// TIA Portal V15.1 export
// export: Created 2024-05-17T05:38:13.9660072Z, ExportSetting WithDefaults, DisplayName Totally Integrated Automation Portal, DisplayVersion V15.1 Update 5, DisplayName TIA Portal Openness, DisplayVersion V15.1 Update 5, DisplayName SINAMICS Startdrive Advanced, DisplayVersion V15.1, DisplayName G130, G150, S120, S150, SINAMICS MV, S210, DisplayVersion V15.1, DisplayName G110M, G120, G120C, G120D, G120P, DisplayVersion V15.1, DisplayName STEP 7 Professional, DisplayVersion V15.1 Update 5, DisplayName STEP 7 Safety, DisplayVersion V15.1, DisplayName WinCC Professional, DisplayVersion V15.1 Update 5, DisplayName SIMATIC Visualization Architect, DisplayVersion V15.1
DATA_BLOCK "_209210ZS01PNIODiag"   // DB324
{ S7_Optimized_Access := 'FALSE' }
AUTHOR : VCC
VERSION : 0.1
// stored: AutoNumber false, DBAccessibleFromOPCUA true, IsOnlyStoredInLoadMemory false, IsWriteProtectedInAS false
   VAR RETAIN
      "AA_209210AS10-JW40" { ExternalAccessible := 'False'; ExternalVisible := 'False'; ExternalWritable := 'False'} : Bool;   // Profinet device don't exist - ET200sp I/O - Busnode 210AS10 - node 40
      "AA_209210AX01-JW41" { ExternalAccessible := 'False'; ExternalVisible := 'False'; ExternalWritable := 'False'} : Bool;   // Profinet device don't exist - ET200sp I/O - Busnode 210AX01 - node 41
      "AA_209210AS11-JW42" { ExternalAccessible := 'False'; ExternalVisible := 'False'; ExternalWritable := 'False'} : Bool;   // Profinet device don't exist - ET200sp I/O - Busnode 210AS11 - node 42
      "AA_209210AX02-JW43" { ExternalAccessible := 'False'; ExternalVisible := 'False'; ExternalWritable := 'False'} : Bool;   // Profinet device don't exist - ET200sp I/O - Busnode 210AX02 - node 43
      "AC_209210CWP10-JX44" { ExternalAccessible := 'False'; ExternalVisible := 'False'; ExternalWritable := 'False'} : Bool;   // Profinet device don't exist - ET200eco I/O - Module 210CWP10 - node 44
      "AC_209210CWP10-JX45" { ExternalAccessible := 'False'; ExternalVisible := 'False'; ExternalWritable := 'False'} : Bool;   // Profinet device don't exist - ET200eco I/O - Module 210CWP10 - node 45
      "AC_209210CWP20-JX46" { ExternalAccessible := 'False'; ExternalVisible := 'False'; ExternalWritable := 'False'} : Bool;   // Profinet device don't exist - ET200eco I/O - Module 210CWP20 - node 46
      "AC_209210CWP20-JX47" { ExternalAccessible := 'False'; ExternalVisible := 'False'; ExternalWritable := 'False'} : Bool;   // Profinet device don't exist - ET200eco I/O - Module 210CWP20 - node 47
      "AA_209210AS20-JW48" { ExternalAccessible := 'False'; ExternalVisible := 'False'; ExternalWritable := 'False'} : Bool;   // Profinet device don't exist - ET200sp I/O - Busnode 210AS20 - node 48
      "AB_209000AK03M1-UE130" { ExternalAccessible := 'False'; ExternalVisible := 'False'; ExternalWritable := 'False'} : Bool;   // Profinet device don't exist - MoviDrive - 210CR21M1 - node 130
      "AB_209000AK03M4-UE131" { ExternalAccessible := 'False'; ExternalVisible := 'False'; ExternalWritable := 'False'} : Bool;   // Profinet device don't exist - MoviDrive - 210CS22M4(Power) - node 131
      "AB_209000AK03M4-UE132" { ExternalAccessible := 'False'; ExternalVisible := 'False'; ExternalWritable := 'False'} : Bool;   // Profinet device don't exist - MoviDrive - 210CS22M4(Brake) - node 132
      "AB_209000AK03M1-UE133" { ExternalAccessible := 'False'; ExternalVisible := 'False'; ExternalWritable := 'False'} : Bool;   // Profinet device don't exist - MoviDrive - 210CR23M1 - node 133
      "AB_209210CHB21M14-UE134" { ExternalAccessible := 'False'; ExternalVisible := 'False'; ExternalWritable := 'False'} : Bool;   // Profinet device don't exist - MoviFit - 210CHB21M14 - node 134
      "AA_209210Field-JW221" { ExternalAccessible := 'False'; ExternalVisible := 'False'; ExternalWritable := 'False'} : Bool;   // Profinet device don't exist - Field Switch - Safety Zone 210 - node 221
      "AA_209210Field-JW231" { ExternalAccessible := 'False'; ExternalVisible := 'False'; ExternalWritable := 'False'} : Bool;   // Profinet device don't exist - Field Switch - Safety Zone 210 - node 231
      "AC_209210AS10-JW40Fault" { ExternalAccessible := 'False'; ExternalVisible := 'False'; ExternalWritable := 'False'} : Bool;   // Faulty profinet device -> For more detail information look for N.A. alarms in the alarmlist - ET200sp I/O - Busnode 210AS10 - node 40
      "AC_209210AX01-JW41Fault" { ExternalAccessible := 'False'; ExternalVisible := 'False'; ExternalWritable := 'False'} : Bool;   // Faulty profinet device -> For more detail information look for N.A. alarms in the alarmlist - ET200sp I/O - Busnode 210AX01 - node 41
      "AC_209210AS11-JW42Fault" { ExternalAccessible := 'False'; ExternalVisible := 'False'; ExternalWritable := 'False'} : Bool;   // Faulty profinet device -> For more detail information look for N.A. alarms in the alarmlist - ET200sp I/O - Busnode 210AS11 - node 42
      "AC_209210AX02-JW43Fault" { ExternalAccessible := 'False'; ExternalVisible := 'False'; ExternalWritable := 'False'} : Bool;   // Faulty profinet device -> For more detail information look for N.A. alarms in the alarmlist - ET200sp I/O - Busnode 210AX02 - node 43
      "AC_209210CWP10-JX44Fault" { ExternalAccessible := 'False'; ExternalVisible := 'False'; ExternalWritable := 'False'} : Bool;   // Faulty profinet device -> For more detail information look for N.A. alarms in the alarmlist - ET200eco I/O - Module 210CWP10 - node 44
      "AC_209210CWP10-JX45Fault" { ExternalAccessible := 'False'; ExternalVisible := 'False'; ExternalWritable := 'False'} : Bool;   // Faulty profinet device -> For more detail information look for N.A. alarms in the alarmlist - ET200eco I/O - Module 210CWP10 - node 45
      "AC_209210CWP20-JX46Fault" { ExternalAccessible := 'False'; ExternalVisible := 'False'; ExternalWritable := 'False'} : Bool;   // Faulty profinet device -> For more detail information look for N.A. alarms in the alarmlist - ET200eco I/O - Module 210CWP20 - node 46
      "AC_209210CWP20-JX47Fault" { ExternalAccessible := 'False'; ExternalVisible := 'False'; ExternalWritable := 'False'} : Bool;   // Faulty profinet device -> For more detail information look for N.A. alarms in the alarmlist - ET200eco I/O - Module 210CWP20 - node 47
      "AC_209210AS20-JW48Fault" { ExternalAccessible := 'False'; ExternalVisible := 'False'; ExternalWritable := 'False'} : Bool;   // Faulty profinet device -> For more detail information look for N.A. alarms in the alarmlist - ET200sp I/O - Busnode 210AS20 - node 48
      "AC_209000AK03M1-UE130Fault" { ExternalAccessible := 'False'; ExternalVisible := 'False'; ExternalWritable := 'False'} : Bool;   // Faulty profinet device -> For more detail information look for N.A. alarms in the alarmlist - MoviDrive - 210CR21M1 - node 130
      "AC_209000AK03M4-UE131Fault" { ExternalAccessible := 'False'; ExternalVisible := 'False'; ExternalWritable := 'False'} : Bool;   // Faulty profinet device -> For more detail information look for N.A. alarms in the alarmlist - MoviDrive - 210CS22M4(Power) - node 131
      "AC_209000AK03M4-UE132Fault" { ExternalAccessible := 'False'; ExternalVisible := 'False'; ExternalWritable := 'False'} : Bool;   // Faulty profinet device -> For more detail information look for N.A. alarms in the alarmlist - MoviDrive - 210CS22M4(Brake) - node 132
      "AC_209000AK03M1-UE133Fault" { ExternalAccessible := 'False'; ExternalVisible := 'False'; ExternalWritable := 'False'} : Bool;   // Faulty profinet device -> For more detail information look for N.A. alarms in the alarmlist - MoviDrive - 210CR23M1 - node 133
      "AC_209210CHB21M14-UE134Fault" { ExternalAccessible := 'False'; ExternalVisible := 'False'; ExternalWritable := 'False'} : Bool;   // Faulty profinet device -> For more detail information look for N.A. alarms in the alarmlist - MoviFit - 210CHB21M14 - node 134
      "AC_209210Field-JW221Fault" { ExternalAccessible := 'False'; ExternalVisible := 'False'; ExternalWritable := 'False'} : Bool;   // Faulty profinet device -> For more detail information look for N.A. alarms in the alarmlist - Field Switch - Safety Zone 210 - node 221
      "AC_209210Field-JW231Fault" { ExternalAccessible := 'False'; ExternalVisible := 'False'; ExternalWritable := 'False'} : Bool;   // Faulty profinet device -> For more detail information look for N.A. alarms in the alarmlist - Field Switch - Safety Zone 210 - node 231
      "209210AS10-JW40AlarmABCondition" { ExternalAccessible := 'False'; ExternalVisible := 'False'; ExternalWritable := 'False'} : Bool;   // Alarm AB condition
      "209210AX01-JW41AlarmABCondition" { ExternalAccessible := 'False'; ExternalVisible := 'False'; ExternalWritable := 'False'} : Bool;   // Alarm AB condition
      "209210AS11-JW42AlarmABCondition" { ExternalAccessible := 'False'; ExternalVisible := 'False'; ExternalWritable := 'False'} : Bool;   // Alarm AB condition
      "209210AX02-JW43AlarmABCondition" { ExternalAccessible := 'False'; ExternalVisible := 'False'; ExternalWritable := 'False'} : Bool;   // Alarm AB condition
      "209210AS20-JW48AlarmABCondition" { ExternalAccessible := 'False'; ExternalVisible := 'False'; ExternalWritable := 'False'} : Bool;   // Alarm AB condition
      "209000AK03M1-UE130AlarmABCondition" { ExternalAccessible := 'False'; ExternalVisible := 'False'; ExternalWritable := 'False'} : Bool;   // Alarm AB condition
      "209000AK03M4-UE131AlarmABCondition" { ExternalAccessible := 'False'; ExternalVisible := 'False'; ExternalWritable := 'False'} : Bool;   // Alarm AB condition
      "209000AK03M4-UE132AlarmABCondition" { ExternalAccessible := 'False'; ExternalVisible := 'False'; ExternalWritable := 'False'} : Bool;   // Alarm AB condition
      "209000AK03M1-UE133AlarmABCondition" { ExternalAccessible := 'False'; ExternalVisible := 'False'; ExternalWritable := 'False'} : Bool;   // Alarm AB condition
      "209210CHB21M14-UE134AlarmABCondition" { ExternalAccessible := 'False'; ExternalVisible := 'False'; ExternalWritable := 'False'} : Bool;   // Alarm AB condition
      "209210Field-JW221AlarmABCondition" { ExternalAccessible := 'False'; ExternalVisible := 'False'; ExternalWritable := 'False'} : Bool;   // Alarm AB condition
      "209210Field-JW231AlarmABCondition" { ExternalAccessible := 'False'; ExternalVisible := 'False'; ExternalWritable := 'False'} : Bool;   // Alarm AB condition
      "H_209210AS10-JW40IAnim" : Word;   // HMI Animation of the icon
      "H_209210AX01-JW41IAnim" : Word;   // HMI Animation of the icon
      "H_209210AS11-JW42IAnim" : Word;   // HMI Animation of the icon
      "H_209210AX02-JW43IAnim" : Word;   // HMI Animation of the icon
      "H_209210CWP10-JX44IAnim" : Word;   // HMI Animation of the icon
      "H_209210CWP10-JX45IAnim" : Word;   // HMI Animation of the icon
      "H_209210CWP20-JX46IAnim" : Word;   // HMI Animation of the icon
      "H_209210CWP20-JX47IAnim" : Word;   // HMI Animation of the icon
      "H_209210AS20-JW48IAnim" : Word;   // HMI Animation of the icon
      "H_209000AK03M1-UE130IAnim" : Word;   // HMI Animation of the icon
      "H_209000AK03M4-UE131IAnim" : Word;   // HMI Animation of the icon
      "H_209000AK03M4-UE132IAnim" : Word;   // HMI Animation of the icon
      "H_209000AK03M1-UE133IAnim" : Word;   // HMI Animation of the icon
      "H_209210CHB21M14-UE134IAnim" : Word;   // HMI Animation of the icon
      "H_209210Field-JW221IAnim" : Word;   // HMI Animation of the icon
      "H_209210Field-JW231IAnim" : Word;   // HMI Animation of the icon
      "H_209210AS10-JW40IAnim2" : Word;   // HMI Animation of the icon
      "H_209210AX01-JW41IAnim2" : Word;   // HMI Animation of the icon
      "H_209210AS11-JW42IAnim2" : Word;   // HMI Animation of the icon
      "H_209210AX02-JW43IAnim2" : Word;   // HMI Animation of the icon
      "H_209210CWP10-JX44IAnim2" : Word;   // HMI Animation of the icon
      "H_209210CWP10-JX45IAnim2" : Word;   // HMI Animation of the icon
      "H_209210CWP20-JX46IAnim2" : Word;   // HMI Animation of the icon
      "H_209210CWP20-JX47IAnim2" : Word;   // HMI Animation of the icon
      "H_209210AS20-JW48IAnim2" : Word;   // HMI Animation of the icon
      "H_209000AK03M1-UE130IAnim2" : Word;   // HMI Animation of the icon
      "H_209000AK03M4-UE131IAnim2" : Word;   // HMI Animation of the icon
      "H_209000AK03M4-UE132IAnim2" : Word;   // HMI Animation of the icon
      "H_209000AK03M1-UE133IAnim2" : Word;   // HMI Animation of the icon
      "H_209210CHB21M14-UE134IAnim2" : Word;   // HMI Animation of the icon
      "H_209210Field-JW221IAnim2" : Word;   // HMI Animation of the icon
      "H_209210Field-JW231IAnim2" : Word;   // HMI Animation of the icon
      H_IAnim : Word;   // Icon Animation / Animation
      H_Anim : Word;   // Animation
      H_DBnr : Int;   // DB number
      AlarmA { ExternalAccessible := 'False'; ExternalVisible := 'False'; ExternalWritable := 'False'} : Bool;   // Summary Alarm A
      AlarmB { ExternalAccessible := 'False'; ExternalVisible := 'False'; ExternalWritable := 'False'} : Bool;   // Summary Alarm B
      AlarmC { ExternalAccessible := 'False'; ExternalVisible := 'False'; ExternalWritable := 'False'} : Bool;   // Summary Alarm C
      AlarmD { ExternalAccessible := 'False'; ExternalVisible := 'False'; ExternalWritable := 'False'} : Bool;   // Summary Alarm D
      AlarmABCondition { ExternalAccessible := 'False'; ExternalVisible := 'False'; ExternalWritable := 'False'} : Bool;   // Alarm AB Condition
   END_VAR
BEGIN
END_DATA_BLOCK
